Fanuc KAREL source: kf00061.compact.KL

PROGRAM KF00061
%STACKSIZE=65535
%PRIORITY=65535
%NOLOCKGROUP
VAR
I : INTEGER
J : INTEGER
X : REAL
Y : REAL
B : BOOLEAN
C : BOOLEAN
TXT : STRING[80]
TXT2 : STRING[80]
AI : ARRAY[4] OF INTEGER
BI : ARRAY[4] OF INTEGER
P : XYZWPR
JP : JOINTPOS9
PF : POSITION
V1 : VECTOR
V2 : VECTOR
STATUS : INTEGER
BEGIN
I=2
X=0.5
Y=1.0
X=ATAN2(X,Y)
END KF00061
